INTERFACE I_Component EXTENDS I_Object

METHOD PUBLIC M_Request : BOOL
VAR_INPUT
	eRequest:	E_Request;
END_VAR
END_METHOD

PROPERTY PUBLIC P_Event : I_Event
GET
END_GET
END_PROPERTY

PROPERTY PUBLIC P_Reflection : I_Reflection
GET
END_GET
END_PROPERTY

PROPERTY PUBLIC P_State : E_State
GET
END_GET
END_PROPERTY

END_INTERFACE

(* stored: Version 1.1.0.1
   Itf I_Component: Id {84a5f8f6-b81b-4747-a25d-2c3abe61b573}
   Method M_Request: Id {5bce4574-fbb8-4134-a60e-e5f2d429768c}
   Property P_Event: Id {b939a253-76b4-0945-2846-e8d6d6fe98d7}
   Get Get: Id {9a694d2d-d968-0612-382b-8a637ec7c25b}
   Property P_Reflection: Id {e4c55aa1-6e83-089d-307d-057e145ff2a0}
   Get Get: Id {57af0f07-74f8-0d86-3b67-d5a15cd0686a}
   Property P_State: Id {9375c264-99fd-089c-38fd-cd77509e54a2}
   Get Get: Id {60f93b25-f1b0-038e-0539-4522cdd6500b} *)
